PROGRAM POU_FaultHandler_Momentary
VAR
	tonTimer: ARRAY[0..100] OF Ton;
	bPowerUp: BOOL;
END_VAR



//------_________________________-----------------------------------------------------------------------------------------------------
//----- Related to System Faults -----------------------------------------------------------------------------------------------------

IF PRG_MasterControl.bPowerUpDone AND NOT bPowerUp THEN
		GVL_Alarms.arrEventFlag[200]:= TRUE;
		bPowerUp:= TRUE;
		tonTimer[0](in:=TRUE, pt:= T#5S);
	ELSIF tonTimer[0].Q THEN
		GVL_Alarms.arrEventFlag[200]:= FALSE;	
END_IF


//*********************************************************END SECTION****************************************************************



//------____________________________--------------------------------------------------------------------------------------------------
//----- Related to Interlock Errors --------------------------------------------------------------------------------------------------




//*********************************************************END SECTION****************************************************************

//------____________________________--------------------------------------------------------------------------------------------------
//----- Related to Process Warnings --------------------------------------------------------------------------------------------------



//*********************************************************END SECTION****************************************************************

END_PROGRAM

(* stored: Version 1.1.0.1, ProductVersion 3.1.4024.12
   POU POU_FaultHandler_Momentary: Id {4873ef46-eff7-47ff-9964-3c64275d0e19}, SpecialFunc None *)
